RoboDK station: workstation_box_pick_place.rdk

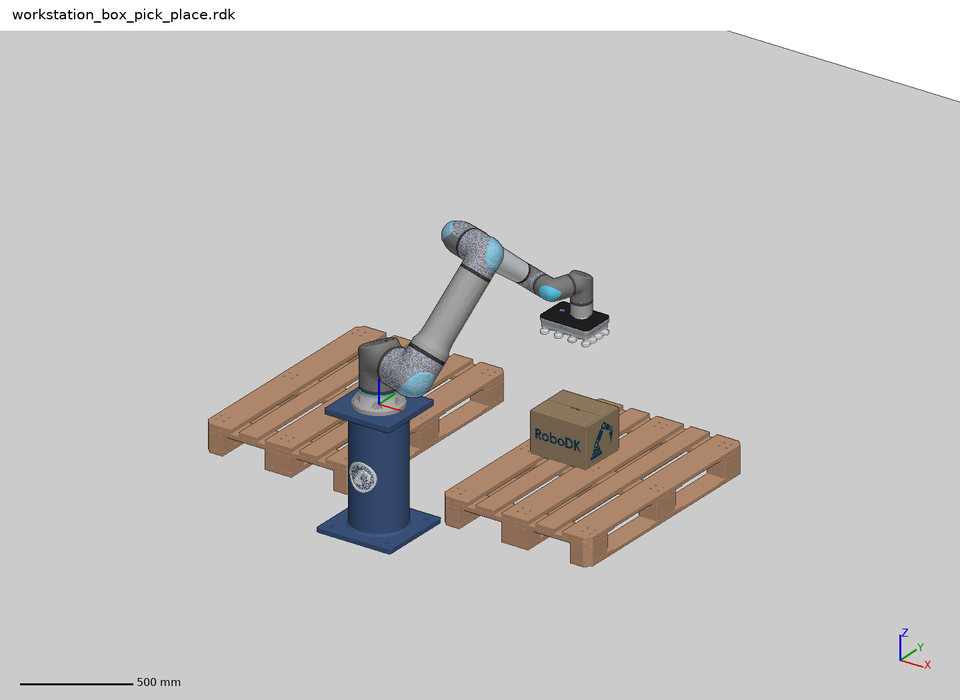
[picture v0: the station drawn from its stored meshes, robots at their saved joint values, targets as dots, program paths as lines]
Station box_pick_plac (saved by RoboDK 5.2.4). Poses are relative to the parent item; angles as X-Y-Z fixed-axis rotations.
  - frame UR30 Base at (0, 0, 610) mm
    - robot UR30 (model UR20): 6 axes
        modified DH rows (alpha deg, a mm, theta deg, d mm): 0, 0, 0, 236.2; 90, 0, -180, 0; 0, 636.8, 0, 0; 0, 505.7, 0, 201.9; -90, 0, 0, 159.4; 90, 0, 0, 154.8
        joint limits [-360, -360, -360, -360, -360, -360] to [360, 360, 360, 360, 360, 360]; home [0, -90, -90, 0, 90, 0]; saved at [70.115, -128.839, -89.791, -51.37, 90, -19.885]
      - tool Tool, TCP at (0, 0, 100) mm
      - tool OnRobot VGP20 Vacuum Gripper, TCP at (-36, 0, 106.49) mm, size 268.4 x 184.1 x 103.7 mm
      - tool OnRobot Quick Tool Changer (Robot), TCP at (0, 0, 12.2) mm, size 71 x 70.9 x 16.1 mm
  - object plane at (0, 0, 0) mm, size 10000 x 10000 x 0 mm, geometry from plane.obj
  - object box at (330, 948.84, 180) mm, rotated rx 0 ry 0 rz -90 deg, size 252 x 305.4 x 216.7 mm, geometry from Box-12x10in-Closed.sld
  - object Pallet 1200x800mm (Transverse) at (-1050, 150, 170) mm, size 800 x 1200 x 144.2 mm, geometry from Pallet-1200x800mm-Transverse.sld
  - object Pallet 1200x800mm (Transverse) at (230, 150, 170) mm, size 800 x 1200 x 144.2 mm, geometry from Pallet-1200x800mm-Transverse.sld
  - object Pedestal H24in (Type 1) at (0, 0, 0) mm, size 400 x 400 x 609.6 mm, geometry from Pedestal-H24in-Type-1.sld
  - program Resert (1 instructions, listed below)

--- program Resert (robot UR30) ---
  Replace box
